# EPICS substitutions: db/PSI/ecmcPSI_TEST_01.substitutions
file "ecmcEcSlave.template"
{
  pattern {}
          {}
}

file "ecmc_analogOutput-chX.template"
{
  pattern {CH_ID, KEY,          sourceName,     EGU, PREC, DRVL, DRVH}
          {01,    ledBlinkRate, ledBlinkRate,   "ms", 0,    0,    0   }
}

file "ecmc_binaryOutput-chX.template"
{
  pattern {CH_ID, KEY,      sourceName, ZNAM, ONAM}
          {01,    ledonoff, ledonoff,   Off,  On  }
}

file "ecmc_analogInputFloat-chX.template"
{
  pattern {CH_ID, KEY,     sourceName, ESLO, EGU, PREC}
          {01,    counter, counter,    1,    "",  3   }
}

file "ecmc_analogInput-chX.template"
{
  pattern {CH_ID, KEY,    sourceName, ESLO, EGU, PREC}
          {01,    uptime, uptime,     1,    "s", 0   }
}
